function_block FB_Syntax_DisableRegions var nA : int; nB      : int; end_var

nA := 1;


{formatting.disable}
nA := 99;
nB := 88;
{formatting.enable}


(* formatting.disable *)
nA := 77;
(* formatting.enable *)
nB := 2;

END_FUNCTION_BLOCK

(* stored: Version 1.1.0.1, ProductVersion 3.1.4024.16
   POU FB_Syntax_DisableRegions: Id {4b840b4c-b961-4dfe-b7a7-f5cf757f38e2}, SpecialFunc None *)
